// TwinCAT 3 PLC project Untitled1
// ProgramVersion: 3.1.4024.0
// libraries:
//   Tc2_MC2, * (Beckhoff Automation GmbH)
//   Tc2_Standard, * (Beckhoff Automation GmbH)
//   Tc2_System, * (Beckhoff Automation GmbH)
//   Tc3_Module, * (Beckhoff Automation GmbH)
// project tree:
//   / PlcTask.TcTTO
//   POUs/ MAIN.TcPOU
// real-time tasks:
//   TASK PlcTask: cycle T#10ms, priority 20, ADS port 350
// motion (NC):
//   TASK NC-Task 1 SAF: cycle T#2ms, priority 4, ADS port 501
//   TASK NC-Task 1 SVB: cycle T#10ms, priority 8, ADS port 511
//   AXIS Axis 1 (id 1)
//     OtherSettings: AllowMotionCmdToSlave=true
//     encoder EncType=1
//     drive DrvType=5
//       Analog: TorqueSetpointScale=10, ScaleFactorActTorque=0.1
//       TimeComp: TaskDelayCycles=1
//     controller CtrType=1
//       CtrPara: PriorControlFactor=1
//         Observer: BandWidth=20
//   AXIS Axis 2 (id 2)
//     OtherSettings: AllowMotionCmdToSlave=true
//     encoder EncType=1
//     drive DrvType=5
//       Analog: TorqueSetpointScale=10, ScaleFactorActTorque=0.1
//       TimeComp: TaskDelayCycles=1
//     controller CtrType=1
//       CtrPara: PriorControlFactor=1
//         Observer: BandWidth=20
//   AXIS Axis 3 (id 3)
//     OtherSettings: AllowMotionCmdToSlave=true
//     encoder EncType=1
//     drive DrvType=5
//       Analog: TorqueSetpointScale=10, ScaleFactorActTorque=0.1
//       TimeComp: TaskDelayCycles=1
//     controller CtrType=1
//       CtrPara: PriorControlFactor=1
//         Observer: BandWidth=20
//   AXIS Axis 4 (id 4)
//     OtherSettings: AllowMotionCmdToSlave=true
//     encoder EncType=1
//     drive DrvType=5
//       Analog: TorqueSetpointScale=10, ScaleFactorActTorque=0.1
//       TimeComp: TaskDelayCycles=1
//     controller CtrType=1
//       CtrPara: PriorControlFactor=1
//         Observer: BandWidth=20
//   AXIS Axis 5 (id 5)
//     OtherSettings: AllowMotionCmdToSlave=true
//     encoder EncType=1
//     drive DrvType=5
//       Analog: TorqueSetpointScale=10, ScaleFactorActTorque=0.1
//       TimeComp: TaskDelayCycles=1
//     controller CtrType=1
//       CtrPara: PriorControlFactor=1
//         Observer: BandWidth=20
// variable links:
//   Untitled1/Untitled1 Instance <-> NC-Task 1 SAF/Axes/Axis 1
//     PlcTask Inputs/MAIN.axis1.NcToPlc <-> Outputs/ToPlc
//     PlcTask Outputs/MAIN.axis1.PlcToNc <-> Inputs/FromPlc
//   Untitled1/Untitled1 Instance <-> NC-Task 1 SAF/Axes/Axis 2
//     PlcTask Inputs/MAIN.axis2.NcToPlc <-> Outputs/ToPlc
//     PlcTask Outputs/MAIN.axis2.PlcToNc <-> Inputs/FromPlc
//   Untitled1/Untitled1 Instance <-> NC-Task 1 SAF/Axes/Axis 3
//     PlcTask Inputs/MAIN.axis3.NcToPlc <-> Outputs/ToPlc
//     PlcTask Outputs/MAIN.axis3.PlcToNc <-> Inputs/FromPlc
//   Untitled1/Untitled1 Instance <-> NC-Task 1 SAF/Axes/Axis 4
//     PlcTask Inputs/MAIN.axis4.NcToPlc <-> Outputs/ToPlc
//     PlcTask Outputs/MAIN.axis4.PlcToNc <-> Inputs/FromPlc
//   Untitled1/Untitled1 Instance <-> NC-Task 1 SAF/Axes/Axis 5
//     PlcTask Inputs/MAIN.axis5.NcToPlc <-> Outputs/ToPlc
//     PlcTask Outputs/MAIN.axis5.PlcToNc <-> Inputs/FromPlc

CONFIGURATION Untitled1
    RESOURCE PLC ON TwinCAT3
        TASK PlcTask(INTERVAL := T#10ms, PRIORITY := 20);
        PROGRAM MAIN WITH PlcTask : MAIN;
    END_RESOURCE
END_CONFIGURATION

// ---- POUs/MAIN.TcPOU
PROGRAM MAIN
VAR
	axis1 					: AXIS_REF;
	axis2 					: AXIS_REF;
	axis3 					: AXIS_REF;
	axis4 					: AXIS_REF;
	axis5 					: AXIS_REF;
	fbPower1 				: MC_Power;
	fbPower2 				: MC_Power;
	fbPower3				: MC_Power;
	fbPower4 				: MC_Power;
	fbPower5 				: MC_Power;
	
	aEnable					: BOOL;
	fb_GearInMultiMaster	: MC_GearInMultiMaster;
	gEbable					: BOOL;
	fbMove 					: MC_MoveAbsolute;
	fbMove2 					: MC_MoveAbsolute;
	fbMove3 					: MC_MoveAbsolute;
	fbMove4 					: MC_MoveAbsolute;
oran 							: DWORD:=2;
	mEnable: BOOL;
END_VAR

//aEnable eksenleri enable etmek için ,gEbable fb_GearInMultiMaster fonksiyon bloğunu çalıştımak için, menable eksenlere hareket verebilmek için
fbPower1(
	Axis:=axis1 , 
	Enable:=aEnable, 
	Enable_Positive:= aEnable, 
	Enable_Negative:=aEnable , 
	Override:=100 );
	
fbPower2(
	Axis:=axis2 , 
	Enable:=aEnable, 
	Enable_Positive:= aEnable, 
	Enable_Negative:=aEnable , 
	Override:=100);
	
fbPower3(
	Axis:=axis3 , 
	Enable:=aEnable, 
	Enable_Positive:= aEnable, 
	Enable_Negative:=aEnable , 
	Override:=100);
	
fbPower4(
	Axis:=axis4 , 
	Enable:=aEnable, 
	Enable_Positive:= aEnable, 
	Enable_Negative:=aEnable , 
	Override:=100);
	
fbPower5(
	Axis:=axis5 , 
	Enable:=aEnable, 
	Enable_Positive:= aEnable, 
	Enable_Negative:=aEnable , 
	Override:=100);
	
	
fb_GearInMultiMaster(
	Master1:= axis1, 
	Master2:= axis2, 
	Master3:= axis3, 
	Master4:= axis4, 
	Slave  := axis5, 
	Enable := gEbable , 
	GearRatio1:= 1, 
	GearRatio2:= 2, 
	GearRatio3:= 3, 
	GearRatio4:= 4);

fbMove(
	Axis:= axis1, 
	Execute:=mEnable , 
	Position:=10 , 
	Velocity:= 10 );
	
fbMove2(
	Axis:= axis2, 
	Execute:=mEnable , 
	Position:=10 , 
	Velocity:= 10 );

fbMove3(
	Axis:= axis3, 
	Execute:=mEnable , 
	Position:=10 , 
	Velocity:= 10  );
	
fbMove4(
	Axis:= axis4, 
	Execute:=mEnable , 
	Position:=10 , 
	Velocity:= 10 );

END_PROGRAM
